# EPICS substitutions: ethmodApp/Db/AKI2C_TMP100.substitutions
file AKI2C_TMP100_dev.template
{
   pattern { P    ,R    ,PORT    ,ADDR     ,TIMEOUT     }
           { $(P) ,$(R) ,$(PORT) ,$(ADDR)  ,$(TIMEOUT)  }
}
